/////////////////////////////////////////////////////////////////////////////////////MACHINE STATUS/////////////////////////////////////////////////////////////////////////////////////
stMachineStatus.bSystemPowerUp 			:= (stMachineStatus.eMachineState = E_MachineState.SYSTEM_POWER_UP);
stMachineStatus.bStopped 				:= (stMachineStatus.eMachineState = E_MachineState.STOPPED);
stMachineStatus.bInitialising 			:= (stMachineStatus.eMachineState = E_MachineState.SYSTEM_INITIALISING);
stMachineStatus.bReadyToStart 			:= (stMachineStatus.eMachineState = E_MachineState.SYSTEM_READY_TO_START);
stMachineStatus.bAutoCycle 				:= (stMachineStatus.eMachineState = E_MachineState.SYSTEM_AUTO_CYCLE);
stMachineStatus.bStopping 				:= (stMachineStatus.eMachineState = E_MachineState.STOPPING);
stMachineStatus.bFault 					:= (stMachineStatus.eMachineState = E_MachineState.FAULT);
stMachineStatus.bManualMode 			:= (stMachineStatus.eMachineState = E_MachineState.MANUAL_MODE);
stMachineStatus.bSafety 				:= (stMachineStatus.eMachineState = E_MachineState.SAFETY);

/////////////////////////////////////////////////////////////////////////////////////FLAGS/////////////////////////////////////////////////////////////////////////////////////
stMasterCtrl.bAllStationsStopped		:= (stCamera.Status.bStopped OR NOT stMACHINE.bVisionTest ) AND (stLeakTesters.Status.bStopped OR NOT stMACHINE.bLeakTest ) AND (stHeightTests.Status.bStopped OR NOT stMACHINE.bHeightTest ) AND stProcessCylinder.Status.bStopped AND stProcessDoor.Status.bStopped AND
										   (NOT stCamera.Status.bBusy OR NOT stMACHINE.bVisionTest ) AND (NOT stLeakTesters.Status.bBusy OR NOT stMACHINE.bLeakTest ) AND (NOT stHeightTests.Status.bBusy OR NOT stMACHINE.bHeightTest ) AND NOT stProcessCylinder.Status.bBusy AND NOT stProcessDoor.Status.bBusy;
										   
stMasterCtrl.bAllStationsReady			:= (stCamera.Status.bReady OR NOT stMACHINE.bVisionTest ) AND (stLeakTesters.Status.bReady OR NOT stMACHINE.bLeakTest ) AND (stHeightTests.Status.bReady OR NOT stMACHINE.bHeightTest ) AND stProcessCylinder.Status.bReady AND stProcessDoor.Status.bReady;
END_ACTION

ACTION b_ACT_ProcessCycle:
/////////////////////////////////////////////////////////////////////////////////////UTILITIES & TRIGGERS/////////////////////////////////////////////////////////////////////////////////////
//ADD REJECT SENSOR FUNCTION. IF PART FAIL WE SHOULD WAIT UNTIL THE OPERATOR LEAVE THE FAIL PART IN THE CONTAINER
tonTakePicture(IN := stCamera.Status.bDone, PT := T#500MS);

ctuRejectPart();
IF eCycleState = E_General_ProcessCycle.RESET_ALL_CMD THEN
	
	ctuRejectPart.RESET							:= TRUE;

ELSE ctuRejectPart.RESET						:= FALSE;	
	
END_IF
IF eCycleState = E_General_ProcessCycle.IDLE THEN
	
	bAutocycleIDLE								:= TRUE;
	
ELSE bAutocycleIDLE								:= FALSE;

END_IF

tonWaitExtendCylidner(IN := eCycleState = E_General_ProcessCycle.PROCESS_FLAGS_DEFINITIONS, PT := T#1S);
tonGettingResults( IN := eCycleState = E_General_ProcessCycle.WAIT_RESULTS, PT := T#100MS);

tonCMD_Done( IN := , PT := T#500MS);
tonSave_Data( IN :=  eCycleState = E_General_ProcessCycle.SAVE_DATA2, PT := T#500MS);
tonResetAllCMD( IN := eCycleState = E_General_ProcessCycle.RESET_ALL_CMD, PT := T#500MS);


tonExecute( IN := 	eCycleState = E_General_ProcessCycle.CLOSE_PROCESS_DOOR OR
					eCycleState = E_General_ProcessCycle.OPEN_PROCESS_DOOR OR
					eCycleState = E_General_ProcessCycle.WAIT_PRE_RETRACT_PROCESS_CYLINDER OR
					eCycleState = E_General_ProcessCycle.EXTEND_PROCESS_CYLINDER OR
					eCycleState = E_General_ProcessCycle.RETRACT_PROCESS_CYLINDER OR
					eCycleState = E_General_ProcessCycle.CAMERA_INSPECTION OR
					eCycleState = E_General_ProcessCycle.LEAK_TESTS OR
					eCycleState = E_General_ProcessCycle.LEAK_TESTS_HEIGHT_TEST OR
					eCycleState = E_General_ProcessCycle.HEIGHT_TEST OR
					eCycleState = E_General_ProcessCycle.WAIT_TO_SAVE_DATA,
					PT := T#500MS);
					
tonCylinderDwell( IN := eCycleState = E_General_ProcessCycle.PRE_RETRACT_PROCESS_CYLINDER, PT := T#250MS);

IF (stMachineStatus.eMachineState <> E_MachineState.SYSTEM_AUTO_CYCLE) THEN
	
	eCycleState												:= E_General_ProcessCycle.RESET_ALL_CMD;

END_IF

rFirstAutoCycle( CLK := stMachineStatus.bAutoCycle);

IF (eCycleState = E_General_ProcessCycle.CAMERA_INSPECTION) OR (eCycleState = E_General_ProcessCycle.LEAK_TESTS) OR
	(eCycleState = E_General_ProcessCycle.LEAK_TESTS_HEIGHT_TEST) OR (eCycleState = E_General_ProcessCycle.HEIGHT_TEST)  THEN
			sMachineMessage						:= 'Inspection in process';

END_IF

IF stMachineStatus.eMachineState <> E_MachineState.SYSTEM_AUTO_CYCLE THEN
	
	MEMSET( destAddr := ADR(stCycleDataNest1), fillByte := 0, n := SIZEOF(stCycleDataNest1));
	MEMSET( destAddr := ADR(stCycleDataNest2), fillByte := 0, n := SIZEOF(stCycleDataNest2));

END_IF

(* Renan Added 10Jul26*)
bPuckLockerEnable := GVL_Master.stMACHINE.bMachine[2] AND GVL_HMI.bPuckLockerGateEnable;
(*\Renan Added 10Jul26*)

(*Renan added - Puck Locker Bug - 08Jul26*)
bPuckLockerReadyToStart := (NOT bPuckLockerEnable) OR (GVL_Stations.stPuckLocker.bPuckDetected AND
							GVL_Stations.stPuckLocker.bPuckLocked AND GVL_Stations.stPuckLocker.eState = E_PuckLockerState.Locked);
(*\Renan added - Puck Locker Bug - 08Jul26*)

(*Renan Added 06Jul26*)
IF bPuckLockerEnable THEN
	GVL_Stations.stPuckLocker.bNestsEmpty := ((NOT bProcessedPart[0]) OR (NOT bPartPresentNest1)) AND ((NOT bProcessedPart[1]) OR (NOT bPartPresentNest2));
ELSE
	GVL_Stations.stPuckLocker.bNestsEmpty := TRUE;
END_IF
(*\Renan Added 06Jul26*)



/////////////////////////////////////////////////////////////////////////////////////CONDITIONS/////////////////////////////////////////////////////////////////////////////////////

(* Renan Added - Buglist n6 - 08Jul26 *)
bNest1StartOK := (NOT bNest1Flag) OR bPartPresentNest1;
bNest2StartOK := (NOT bNest2Flag) OR bPartPresentNest2;
(*\Renan Added - Buglist n6 - 08Jul26 *)

bStartProcessCondition := bTwoHandsSignal AND bPartPresentNest1 AND bPartPresentNest2 AND (bNest1Flag OR bNest2Flag);

IF rFirstAutoCycle.Q THEN
	eCycleState												:= E_General_ProcessCycle.RESET_ALL_CMD;
END_IF


CASE eCycleState OF
	
E_General_ProcessCycle.RESET_ALL_CMD:

				stProcessDoor.CMD.ProcessDoorCMD.OpenDoor						:= FALSE;
				stProcessDoor.CMD.ProcessDoorCMD.CloseDoor						:= FALSE;
				stProcessDoor.CMD.bExecute										:= FALSE;
				
				stProcessCylinder.CMD.ProcessCylinderCMD.ExtendCylinder1		:= FALSE;
				stProcessCylinder.CMD.ProcessCylinderCMD.RetractCylinder1		:= FALSE;
				stProcessCylinder.CMD.bExecute									:= FALSE;
				
				stLeakTesters.CMD.LeakTestersCMD.RunLeakTester1					:= FALSE;
				stLeakTesters.CMD.LeakTestersCMD.RunLeakTester2					:= FALSE;
				stLeakTesters.CMD.bExecute										:= FALSE;
				
				stHeightTests.CMD.HeightTest_CMD.Measurement1					:= FALSE;
				stHeightTests.CMD.HeightTest_CMD.Measurement2					:= FALSE;
				stHeightTests.CMD.bExecute										:= FALSE;
				
				stCamera.CMD.bExecute											:= FALSE;
				
				bVisionProcessDoneFlag											:= FALSE;
				
				bWriteNest1														:= FALSE;
				bWriteNest2														:= FALSE;
				bRejectPartDialog[0]											:= FALSE;
				bRejectPartDialog[1]											:= FALSE;
				bRejectPartFault												:= FALSE;
				
				bProcessedPart[0]												:= FALSE;
				bProcessedPart[1]												:= FALSE;
			
				//add reset command to reset all cycle data
				
				IF tonResetAllCMD.Q AND stMachineStatus.bAutoCycle THEN
					eCycleState								:= E_General_ProcessCycle.IDLE;						
				END_IF
	
E_General_ProcessCycle.IDLE:

				//start cycle
				IF bStartProcessCondition AND bPartPresent[0] AND bPartPresent[1] AND bPuckLockerReadyToStart THEN (*Renan added - Puck Locker Bug - 08Jul26*) //Original: IF bStartProcessCondition AND NOT bProcessedPart[0] AND NOT bProcessedPart[1] THEN
					
					MEMSET( destAddr := ADR(stCycleDataNest1), fillByte := 0, n := SIZEOF(stCycleDataNest1));
					MEMSET( destAddr := ADR(stCycleDataNest2), fillByte := 0, n := SIZEOF(stCycleDataNest2));
					
					IF bNest1Flag THEN
						
						bProcessedPart[0]					:= bPartPresentNest1;
						
					END_IF
					
					IF bNest2Flag THEN
						
						bProcessedPart[1]					:= bPartPresentNest2;
						
					END_IF
					
					eCycleState								:= E_General_ProcessCycle.CLOSE_PROCESS_DOOR;
					
				END_IF
				
				IF bPuckLockerEnable AND NOT bPuckLockerReadyToStart AND NOT bProcessedPart[0] AND NOT bProcessedPart[1] THEN
				
					IF NOT GVL_Stations.stPuckLocker.bPuckDetected THEN
						
						sMachineMessage 		:= 'Insert puck into locker to continue';
						
					ELSE
						
						sMachineMessage := 'Waiting for puck locker to lock puck';
						
					END_IF					
				
				ELSIF  bPuckLockerReadyToStart AND bPartPresent[0] AND bPartPresent[1] THEN
					
					sMachineMessage := 'trigger both safety buttons to start cycle';
					
				ELSIF bPuckLockerReadyToStart AND ( NOT bPartPresent[0] AND NOT bPartPresent[1]) THEN
					
					sMachineMessage 			:= 'Place parts to continue';
					
				ELSIF bPuckLockerReadyToStart AND ( bPartPresent[0] AND NOT bPartPresent[1]) THEN
					
					sMachineMessage 			:= 'Place part in nest 2 to continue';
				
				ELSIF bPuckLockerReadyToStart AND ( NOT bPartPresent[0] AND bPartPresent[1]) THEN
					
					sMachineMessage 			:= 'Place part in nest 1 to continue';
					
				END_IF
			
E_General_ProcessCycle.CLOSE_PROCESS_DOOR:

				stProcessDoor.CMD.ProcessDoorCMD.CloseDoor	:= TRUE;
				stProcessDoor.CMD.bExecute					:= TRUE;
				
				IF tonExecute.Q THEN
					eCycleState								:= E_General_ProcessCycle.WAIT_CLOSE_PROCESS_DOOR;	
				END_IF

E_General_ProcessCycle.WAIT_CLOSE_PROCESS_DOOR:
				
				IF stProcessDoor.Status.bDone THEN
				stProcessDoor.CMD.ProcessDoorCMD.CloseDoor	:= FALSE;
				stProcessDoor.CMD.bExecute					:= FALSE;
				stProcessDoor.CMD.bAcknowledge				:= TRUE;
				eCycleState									:= E_General_ProcessCycle.PROCESS_FLAGS_DEFINITIONS;
				END_IF
				
E_General_ProcessCycle.PROCESS_FLAGS_DEFINITIONS:
				
				
				IF stMACHINE.bVisionTest THEN
					
					IF bVisionProcessDoneFlag THEN
						
						eCycleState							:= E_General_ProcessCycle.PRE_RETRACT_PROCESS_CYLINDER; //Renan changed - Buglist n13 08Jul26 | Original: \\E_General_ProcessCycle.EXTEND_PROCESS_CYLINDER;
					ELSE eCycleState						:= E_General_ProcessCycle.CAMERA_INSPECTION;
						
					END_IF
				ELSIF tonWaitExtendCylidner.Q AND NOT stMACHINE.bVisionTest THEN

					eCycleState							:= E_General_ProcessCycle.PRE_RETRACT_PROCESS_CYLINDER; //Renan changed - Buglist n13 08Jul26 | Original: \\E_General_ProcessCycle.EXTEND_PROCESS_CYLINDER;
					
				END_IF
				
(* Renan added - Buglist n13 - 08Jul26 *)				
E_General_ProcessCycle.PRE_RETRACT_PROCESS_CYLINDER:		

				stProcessCylinder.CMD.ProcessCylinderCMD.RetractCylinder1		:= TRUE;	
				stProcessCylinder.CMD.bExecute			:= TRUE;
				
				IF tonCylinderDwell.Q THEN
					eCycleState							:= E_General_ProcessCycle.WAIT_PRE_RETRACT_PROCESS_CYLINDER;	
				END_IF

E_General_ProcessCycle.WAIT_PRE_RETRACT_PROCESS_CYLINDER:

				IF 	stProcessCylinder.Status.bDone OR stProcessCylinder.Status.bReady THEN
					
					stProcessCylinder.CMD.ProcessCylinderCMD.RetractCylinder1		:= FALSE;
					stProcessCylinder.CMD.bExecute		:= FALSE;
					stProcessCylinder.CMD.bAcknowledge	:= TRUE;
					
					IF tonExecute.Q THEN
						eCycleState							:= E_General_ProcessCycle.EXTEND_PROCESS_CYLINDER;
					END_IF	
				END_IF
(*\Renan added - Buglist n13 - 08Jul26 *)

E_General_ProcessCycle.EXTEND_PROCESS_CYLINDER:
				
						
				stProcessCylinder.CMD.ProcessCylinderCMD.ExtendCylinder1		:= TRUE;
				stProcessCylinder.CMD.bExecute		:= TRUE;
	
				IF tonExecute.Q THEN
					eCycleState								:= E_General_ProcessCycle.WAIT_EXTEND_PROCESS_CYLINDER;	
				END_IF

E_General_ProcessCycle.WAIT_EXTEND_PROCESS_CYLINDER:
			
				IF stProcessCylinder.Status.bDone THEN
					
					stProcessCylinder.CMD.ProcessCylinderCMD.ExtendCylinder1		:= FALSE;
					stProcessCylinder.CMD.bExecute			:= FALSE;
					stProcessCylinder.CMD.bAcknowledge		:= TRUE;
						
					IF stMACHINE.bHeightTest AND stMACHINE.bLeakTest THEN
						
						eCycleState							:= E_General_ProcessCycle.LEAK_TESTS_HEIGHT_TEST;	
						
					ELSIF 	stMACHINE.bHeightTest AND NOT stMACHINE.bLeakTest  THEN
						
						eCycleState							:= E_General_ProcessCycle.HEIGHT_TEST;
					
					ELSIF 	NOT stMACHINE.bHeightTest AND stMACHINE.bLeakTest  THEN
						
						eCycleState							:= E_General_ProcessCycle.LEAK_TESTS;
					END_IF
					
				END_IF

E_General_ProcessCycle.LEAK_TESTS_HEIGHT_TEST:
				
							
				stLeakTesters.CMD.LeakTestersCMD.RunLeakTester1						:= bNest1Flag;
				stLeakTesters.CMD.LeakTestersCMD.RunLeakTester2						:= bNest2Flag;
				stHeightTests.CMD.HeightTest_CMD.Measurement1						:= bNest1Flag;
				stHeightTests.CMD.HeightTest_CMD.Measurement2						:= bNest2Flag;
				stLeakTesters.CMD.bExecute					:= TRUE;
				stHeightTests.CMD.bExecute					:= TRUE;
							
				IF tonExecute.Q THEN
					eCycleState								:= E_General_ProcessCycle.WAIT_LEAK_TEST_HEIGHT_TEST;	
				END_IF

E_General_ProcessCycle.WAIT_LEAK_TEST_HEIGHT_TEST:
					
					IF stLeakTesters.Status.bDone AND stHeightTests.Status.bDone THEN
						
						stLeakTesters.CMD.LeakTestersCMD.RunLeakTester1				:= FALSE;
						stLeakTesters.CMD.LeakTestersCMD.RunLeakTester2				:= FALSE;
						stHeightTests.CMD.HeightTest_CMD.Measurement1				:= FALSE;
						stHeightTests.CMD.HeightTest_CMD.Measurement2				:= FALSE;
						stLeakTesters.CMD.bExecute			:= FALSE;
						stHeightTests.CMD.bExecute			:= FALSE;
						stLeakTesters.CMD.bAcknowledge		:= TRUE;
						stHeightTests.CMD.bAcknowledge		:= TRUE;
						eCycleState							:= E_General_ProcessCycle.WAIT_RESULTS;
						
					END_IF				   

E_General_ProcessCycle.HEIGHT_TEST:

				stHeightTests.CMD.HeightTest_CMD.Measurement1				 		:= bNest1Flag;
				stHeightTests.CMD.HeightTest_CMD.Measurement2				 		:= bNest2Flag;
				stHeightTests.CMD.bExecute					:= TRUE;
					
				IF tonExecute.Q THEN
					eCycleState								:= E_General_ProcessCycle.WAIT_HEIGHT_TEST;	
				END_IF

E_General_ProcessCycle.WAIT_HEIGHT_TEST:

				IF stHeightTests.Status.bDone THEN
					
					stHeightTests.CMD.HeightTest_CMD.Measurement1				 	:= FALSE;
					stHeightTests.CMD.HeightTest_CMD.Measurement2				 	:= FALSE;
					stHeightTests.CMD.bExecute										:= FALSE;
					stHeightTests.CMD.bAcknowledge 			:= TRUE;	
					eCycleState								:= E_General_ProcessCycle.WAIT_RESULTS;
					
				END_IF

E_General_ProcessCycle.LEAK_TESTS:

				stLeakTesters.CMD.LeakTestersCMD.RunLeakTester1						:= bNest1Flag;
				stLeakTesters.CMD.LeakTestersCMD.RunLeakTester2						:= bNest2Flag;
				stLeakTesters.CMD.bExecute					:= TRUE;
				
				IF tonExecute.Q THEN
					eCycleState								:= E_General_ProcessCycle.WAIT_LEAK_TEST;	
				END_IF

E_General_ProcessCycle.WAIT_LEAK_TEST:

				IF stLeakTesters.Status.bDone THEN
					
					stLeakTesters.CMD.bExecute										:= FALSE;
					stLeakTesters.CMD.LeakTestersCMD.RunLeakTester1				 	:= FALSE;
					stLeakTesters.CMD.LeakTestersCMD.RunLeakTester2				 	:= FALSE;
					stLeakTesters.CMD.bAcknowledge 			:= TRUE;	
					eCycleState								:= E_General_ProcessCycle.WAIT_RESULTS;
					
				END_IF
				
E_General_ProcessCycle.CAMERA_INSPECTION:
				
				stCamera.CMD.bExecute						:= TRUE;
				stCamera.CMD.CameraCMD.Inspect1				:= bNest1Flag;
				stCamera.CMD.CameraCMD.Inspect2				:= bNest2Flag;
				
				IF tonExecute.Q THEN
					eCycleState								:= E_General_ProcessCycle.WAIT_CAMERA;	
				END_IF
				
E_General_ProcessCycle.WAIT_CAMERA:

				IF  tonTakePicture.Q THEN
					
					stCamera.CMD.bExecute					:= FALSE;
					bVisionProcessDoneFlag					:= TRUE;
					stCamera.CMD.bAcknowledge				:= TRUE;
					eCycleState								:= E_General_ProcessCycle.PROCESS_FLAGS_DEFINITIONS;
				
				END_IF
				
E_General_ProcessCycle.WAIT_RESULTS:

				IF tonGettingResults.Q THEN
					
					eCycleState									:= E_General_ProcessCycle.RESULTS;
					
				END_IF


E_General_ProcessCycle.RESULTS:

				
					
					IF bProcessedPart[0] THEN
					
						IF  (stCycleDataNest1.Camera_Pass OR NOT stMACHINE.bVisionTest) AND   (stCycleDataNest1.LeakTest_Pass OR NOT stMACHINE.bLeakTest)
				 			AND   (stCycleDataNest1.HeightTest_Pass OR NOT stMACHINE.bHeightTest) THEN	
				
							stCycleDataNest1.bPass				:= TRUE;
							stCycleDataNest1.bFail				:= FALSE;
				
						ELSE stCycleDataNest1.bFail				:= TRUE;
							stCycleDataNest1.bPass				:= FALSE;
				
						END_IF
					
					END_IF
				
					IF bProcessedPart[1] THEN
					
						IF  (stCycleDataNest2.Camera_Pass OR NOT stMACHINE.bVisionTest) AND   (stCycleDataNest2.LeakTest_Pass OR NOT stMACHINE.bLeakTest)
				 			AND   (stCycleDataNest2.HeightTest_Pass OR NOT stMACHINE.bHeightTest) THEN	
				
							stCycleDataNest2.bPass				:= TRUE;
							stCycleDataNest2.bFail				:= FALSE;
				
						ELSE stCycleDataNest2.bFail				:= TRUE;
							stCycleDataNest2.bPass				:= FALSE;
				
						END_IF
					
					END_IF
					
				
				
				
				
				stCycleDataNest1.sTime						:= sSystemTime;
				stCycleDataNest1.sDate						:= sSystemDate;
				stCycleDataNest2.sTime						:= sSystemTime;
				stCycleDataNest2.sDate						:= sSystemDate;
					
				eCycleState								:= E_General_ProcessCycle.WAIT_TO_SAVE_DATA;
									
E_General_ProcessCycle.WAIT_TO_SAVE_DATA:
				
				IF tonExecute.Q THEN
					eCycleState								:= E_General_ProcessCycle.SAVE_DATA;	
				END_IF

E_General_ProcessCycle.SAVE_DATA:

				IF bProcessedPart[0] THEN
					
					FOR i := 199 TO 0 BY -1 DO
						aDataHistoryNest1[i+1] 						:= aDataHistoryNest1[i];
					END_FOR
				
				END_IF
				
				IF bProcessedPart[1] THEN
					
					FOR i := 199 TO 0 BY -1 DO
						aDataHistoryNest2[i+1] 						:= aDataHistoryNest2[i];
					END_FOR
				
				END_IF		
			
				eCycleState									:= E_General_ProcessCycle.SAVE_DATA2;
					
E_General_ProcessCycle.SAVE_DATA2:	
				
				
				c_ACT_SaveData();	
				
				
					
				eCycleState									:= E_General_ProcessCycle.CSV_NEST1;
				
				
E_General_ProcessCycle.CSV_NEST1:

				IF bProcessedPart[0] THEN
					
					bWriteNest1								:= TRUE;
					
					IF bCSVDone OR bCSVError THEN
						
						eCycleState							:= E_General_ProcessCycle.CSV_NEST2;
						bWriteNest1							:= FALSE;
						bCSVError							:= FALSE;
						
					END_IF
				ELSE eCycleState							:= E_General_ProcessCycle.CSV_NEST2;				
					
				END_IF
			
				
E_General_ProcessCycle.CSV_NEST2:

				IF bCSVDone THEN
					
						bWriteNest2							:= FALSE;
						eCycleState							:= E_General_ProcessCycle.RETRACT_PROCESS_CYLINDER;	
	
				END_IF

				IF bProcessedPart[1] AND  bCSVReady AND NOT bCSVDone AND NOT bCSVError THEN
				
						bWriteNest2							:= TRUE;

				ELSIF NOT bProcessedPart[1] OR bCSVError THEN

						 eCycleState						:= E_General_ProcessCycle.RETRACT_PROCESS_CYLINDER;
						 bCSVError							:= FALSE;
						 
				END_IF
				
				
					
				
E_General_ProcessCycle.RETRACT_PROCESS_CYLINDER:
						
				stProcessCylinder.CMD.ProcessCylinderCMD.RetractCylinder1		:= TRUE;	
				stProcessCylinder.CMD.bExecute			:= TRUE;
				
				IF tonExecute.Q THEN
					eCycleState							:= E_General_ProcessCycle.WAIT_RETRACT_PROCESS_CYLINDER;	
				END_IF

E_General_ProcessCycle.WAIT_RETRACT_PROCESS_CYLINDER:

				IF 	stProcessCylinder.Status.bDone THEN
					
					stProcessCylinder.CMD.ProcessCylinderCMD.RetractCylinder1		:= FALSE;
					stProcessCylinder.CMD.bExecute		:= FALSE;
					stProcessCylinder.CMD.bAcknowledge	:= TRUE;
					
					IF NOT bEmptyRejectChute THEN

						eCycleState							:= E_General_ProcessCycle.OPEN_PROCESS_DOOR;
					
					ELSE eCycleState							:= E_General_ProcessCycle.REJECT_CHUTE_FULL; 
					
					END_IF
					
				END_IF
		
E_General_ProcessCycle.REJECT_CHUTE_FULL:

				sMachineMessage									:= 'Waiting for Reject chute empty';

				IF NOT bEmptyRejectChute THEN
					
						sMachineMessage							:= '';
						eCycleState								:= E_General_ProcessCycle.OPEN_PROCESS_DOOR;
				
				END_IF	
		
E_General_ProcessCycle.OPEN_PROCESS_DOOR:

				stProcessDoor.CMD.ProcessDoorCMD.OpenDoor							:= TRUE;
				stProcessDoor.CMD.bExecute				:= TRUE;
				
				IF tonExecute.Q THEN
					eCycleState							:= E_General_ProcessCycle.WAIT_OPEN_PROCESS_DOOR;	
				END_IF

E_General_ProcessCycle.WAIT_OPEN_PROCESS_DOOR:

				IF 	stProcessDoor.Status.bDone THEN
					
					stProcessDoor.CMD.ProcessDoorCMD.OpenDoor						:= FALSE;
					stProcessDoor.CMD.bExecute			:= FALSE;
					stProcessDoor.CMD.bAcknowledge		:= TRUE;
					
					eCycleState							:= E_General_ProcessCycle.PUCK_DEFINITION;
					
				END_IF
				
E_General_ProcessCycle.PUCK_DEFINITION:
		
				(* Renan Added - Buglist n6 - 08Jul26 *)
				bCycleHasFailure := (bProcessedPart[0] AND stCycleDataNest1.bFail) OR (bProcessedPart[1] AND stCycleDataNest2.bFail);

				bCycleAllProcessedPass := (bProcessedPart[0] OR bProcessedPart[1]) AND ((NOT bProcessedPart[0]) OR stCycleDataNest1.bPass) AND ((NOT bProcessedPart[1]) OR stCycleDataNest2.bPass);
					(*\Renan Added - Buglist n6 - 08Jul26 *)
					
					(* Renan Added 10Jul26 - Puck Locker *)
				IF bPuckLockerEnable AND bCycleAllProcessedPass THEN
					
					GVL_Stations.stPuckLocker.nRequestedRelease := USINT#0;
					
					IF bProcessedPart[0] AND stCycleDataNest1.bPass THEN
						
						GVL_Stations.stPuckLocker.nRequestedRelease := GVL_Stations.stPuckLocker.nRequestedRelease + USINT#1;
						
					END_IF
					
					IF bProcessedPart[1] AND stCycleDataNest2.bPass THEN
						
						GVL_Stations.stPuckLocker.nRequestedRelease := GVL_Stations.stPuckLocker.nRequestedRelease + USINT#1;
							
					END_IF
					
					GVL_Stations.stPuckLocker.bApplyDisposition := TRUE;
					
				END_IF
				
				
				IF bCycleHasFailure THEN //Bugfix 08Jul26
					
					eCycleState								:= E_General_ProcessCycle.WAIT_REJECT_PART;
					
				ELSIF bCycleAllProcessedPass THEN //Bugfix 08Jul26

					eCycleState								:= E_General_ProcessCycle.NEST_CLEARING;
						
				END_IF		
			
E_General_ProcessCycle.WAIT_REJECT_PART:
					
				ctuRejectPart.CU 								:= rRejectSensor.Q;				

				IF stCycleDataNest1.bFail AND NOT stCycleDataNest2.bFail THEN
					
					sMachineMessage												:= 'REMOVE PART FROM NEST 1 AND PUT IN REJECT CHUTE';
					
					IF ctuRejectPart.CV > 0 AND NOT bPartPresentNest1 AND (bPartPresentNest2 OR NOT bProcessedPart[1])  THEN
						
						(* Renan Added 10Jul26 - Puck Locker *)
						IF bPuckLockerEnable THEN
							GVL_Stations.stPuckLocker.nRequestedRelease 		:= USINT#1;
							GVL_Stations.stPuckLocker.bApplyDisposition 		:= TRUE;
						END_IF
						(*\Renan Added 10Jul26 - Puck Locker *)
						
						eCycleState												:= E_General_ProcessCycle.NEST_CLEARING;
						
					ELSIF ctuRejectPart.CV > 0 AND (bPartPresentNest1 OR (NOT bPartPresentNest2 AND bProcessedPart[1])) THEN
						
						bRejectPartFault										:= TRUE; 
					
					END_IF
					
					IF NOT bPartPresentNest2 AND bProcessedPart[1] THEN
						
						bRejectPartDialog[0]									:= TRUE;		
						sMachineMessage											:= 'WRONG PART TAKEN';
						
					ELSIF  bPartPresentNest2 THEN
						
						bRejectPartDialog[0]									:= FALSE;
						
					END_IF					
					
				ELSIF NOT stCycleDataNest1.bFail AND stCycleDataNest2.bFail THEN
					
					sMachineMessage												:= 'REMOVE PART FROM NEST 2 AND PUT IN REJECT CHUTE';
					
					IF ctuRejectPart.CV > 0 AND NOT bPartPresentNest2 AND (bPartPresentNest1 OR NOT bProcessedPart[0])  THEN
						
						(* Renan Added 10Jul26 - Puck Locker *)
						IF bPuckLockerEnable THEN
							GVL_Stations.stPuckLocker.nRequestedRelease 		:= USINT#1;
							GVL_Stations.stPuckLocker.bApplyDisposition 		:= TRUE;
						END_IF
						(*\Renan Added 10Jul26 - Puck Locker *)
						
						
						eCycleState												:= E_General_ProcessCycle.NEST_CLEARING;
						
					ELSIF ctuRejectPart.CV > 0 AND (bPartPresentNest1 OR (NOT bPartPresentNest1 AND bProcessedPart[0])) THEN
						
						bRejectPartFault										:= TRUE; 
					
					END_IF
					
					IF NOT bPartPresentNest1 AND bProcessedPart[0] THEN
						
						bRejectPartDialog[1]									:= TRUE;		
						sMachineMessage											:= 'WRONG PART TAKEN';
						
					ELSIF  bPartPresentNest1 THEN
						
						bRejectPartDialog[1]									:= FALSE;
						
					END_IF
				
				ELSIF stCycleDataNest1.bFail AND stCycleDataNest2.bFail THEN
					
					IF ctuRejectPart.CV > 1 AND NOT bPartPresentNest1 AND NOT bPartPresentNest2 THEN
						
						(* Renan Added 10Jul26 - Puck Locker *)
						IF bPuckLockerEnable THEN
							GVL_Stations.stPuckLocker.nRequestedRelease 		:= USINT#0;
							GVL_Stations.stPuckLocker.bApplyDisposition 		:= TRUE;
						END_IF
						(*\Renan Added 10Jul26 - Puck Locker *)
						
						eCycleState												:= E_General_ProcessCycle.NEST_CLEARING;
					
					ELSIF ctuRejectPart.CV > 1 AND ( bPartPresentNest1 OR bPartPresentNest2) THEN
						
						bRejectPartFault										:= TRUE; 		
					
					END_IF;
					
					sMachineMessage												:= 'REMOVE PART FROM BOTH NESTS AND PUT IN REJECT CHUTE';
					
				END_IF
				
E_General_ProcessCycle.NEST_CLEARING:
				
				IF bPuckLockerEnable AND GVL_Stations.stPuckLocker.eState = E_PuckLockerState.WaitingForNestsEmpty THEN
				
					IF (bPartPresentNest1 AND bNest1Flag) OR (bPartPresentNest2 AND bNest2Flag) THEN
						
						sMachineMessage 										:= 'Remove parts from nests to release puck';
						
					ELSE
						
						sMachineMessage 										:= 'Waiting for puck to be released';
						
					END_IF
				
				ELSIF (bPartPresentNest1 AND bNest1Flag) AND NOT (bPartPresentNest2 AND bNest2Flag)  THEN
					
					IF bPuckLockerEnable THEN
						
						sMachineMessage 										:= 'Remove processed part from nest 1 to release puck';
						
					ELSE
						
						sMachineMessage 										:= 'Remove Processed part from nest 1';
						
					END_IF
					
				ELSIF NOT (bPartPresentNest1 AND bNest1Flag) AND (bPartPresentNest2 AND bNest2Flag)  THEN 
					
					IF bPuckLockerEnable THEN
						
						sMachineMessage 										:= 'Remove processed part from nest 2 to release puck';
						
					ELSE
						
						sMachineMessage 										:= 'Remove Processed part from nest 2';
						
					END_IF
					
				ELSIF (bPartPresentNest1 AND bNest1Flag) AND (bPartPresentNest2 AND bNest2Flag) THEN 
					
					IF bPuckLockerEnable THEN
						
						sMachineMessage 										:= 'Remove processed parts to release puck';
						
					ELSE
						
						sMachineMessage 										:= 'Remove Processed parts';
						
					END_IF
					
				ELSIF (NOT bPartPresentNest1 OR NOT bNest1Flag) AND (NOT bPartPresentNest2 OR NOT bNest2Flag)  THEN
					
					sMachineMessage 											:= '';
					eCycleState													:= E_General_ProcessCycle.RESET_ALL_CMD;
									
				END_IF
				
END_CASE
END_ACTION

ACTION c_ACT_SaveData:

//SAVING NEST 1 DATA
IF bProcessedPart[0] THEN
	
	stCycleDataNest1.sDistance1				:= REAL_TO_STRING(stCycleDataNest1.HeightTest_anDistancesResult[1]);
	stCycleDataNest1.sDistance2				:= REAL_TO_STRING(stCycleDataNest1.HeightTest_anDistancesResult[2]);
	stCycleDataNest1.sDistance3				:= REAL_TO_STRING(stCycleDataNest1.HeightTest_anDistancesResult[3]);
	
	stCycleDataNest1.sSetpoint1				:= REAL_TO_STRING(stCycleDataNest1.HeightTest_anSetPoint[1]);
	stCycleDataNest1.sSetpoint2				:= REAL_TO_STRING(stCycleDataNest1.HeightTest_anSetPoint[2]);
	stCycleDataNest1.sSetpoint3				:= REAL_TO_STRING(stCycleDataNest1.HeightTest_anSetPoint[3]);
	
	IF stCycleDataNest1.bPass THEN
	
		stCycleDataNest1.sGeneralResult			:= 'PASS';

	ELSIF stCycleDataNest1.bFail THEN
	
		stCycleDataNest1.sGeneralResult			:= 'FAIL';

	END_IF
	


	IF stCycleDataNest1.Camera_Pass THEN
	
		stCycleDataNest1.sCameraResult			:= 'PASS';

	ELSIF stCycleDataNest1.Camera_Fail THEN
	
		stCycleDataNest1.sCameraResult			:= 'FAIL';

	END_IF

	IF stCycleDataNest1.HeightTest_Pass THEN
	
		stCycleDataNest1.sHeightTestResult		:= 'PASS';
	
	ELSIF stCycleDataNest1.HeightTest_Fail THEN
	
		stCycleDataNest1.sHeightTestResult		:= 'FAIL';
	
	END_IF



	IF stCycleDataNest1.LeakTest_Pass THEN
	
		stCycleDataNest1.sLeakTesterResult		:= 'PASS';

	ELSIF stCycleDataNest1.LeakTest_Fail THEN
	
		stCycleDataNest1.sLeakTesterResult		:= 'FAIL';
	
	END_IF
	
	aDataHistoryNest1[0]						:= stCycleDataNest1;
	
END_IF;
	

//SAVING NEST 2 DATA

IF bProcessedPart[1] THEN
	
	stCycleDataNest2.sDistance1				:= REAL_TO_STRING(stCycleDataNest2.HeightTest_anDistancesResult[1]);
	stCycleDataNest2.sDistance2				:= REAL_TO_STRING(stCycleDataNest2.HeightTest_anDistancesResult[2]);
	stCycleDataNest2.sDistance3				:= REAL_TO_STRING(stCycleDataNest2.HeightTest_anDistancesResult[3]);
	
	stCycleDataNest2.sSetpoint1				:= REAL_TO_STRING(stCycleDataNest2.HeightTest_anSetPoint[1]);
	stCycleDataNest2.sSetpoint2				:= REAL_TO_STRING(stCycleDataNest2.HeightTest_anSetPoint[2]);
	stCycleDataNest2.sSetpoint3				:= REAL_TO_STRING(stCycleDataNest2.HeightTest_anSetPoint[3]);
	
	IF stCycleDataNest2.bPass THEN
	
		stCycleDataNest2.sGeneralResult			:= 'PASS';

	ELSIF stCycleDataNest2.bFail THEN
	
		stCycleDataNest2.sGeneralResult			:= 'FAIL';

	END_IF
	


	IF stCycleDataNest2.Camera_Pass THEN
	
		stCycleDataNest2.sCameraResult			:= 'PASS';

	ELSIF stCycleDataNest2.Camera_Fail THEN
	
		stCycleDataNest2.sCameraResult			:= 'FAIL';

	END_IF

	IF stCycleDataNest2.HeightTest_Pass THEN
	
		stCycleDataNest2.sHeightTestResult		:= 'PASS';
	
	ELSIF stCycleDataNest2.HeightTest_Fail THEN
	
		stCycleDataNest2.sHeightTestResult		:= 'FAIL';
	
	END_IF



	IF stCycleDataNest2.LeakTest_Pass THEN
	
		stCycleDataNest2.sLeakTesterResult		:= 'PASS';

	ELSIF stCycleDataNest2.LeakTest_Fail THEN
	
		stCycleDataNest2.sLeakTesterResult		:= 'FAIL';
	
	END_IF
	
	aDataHistoryNest2[0]						:= stCycleDataNest2;
	
END_IF
END_ACTION

ACTION d_ACT_IO:
//INPUTS

bPartPresentNest1					:= dw_T08_EL1809.iPartPresentNest1;
bPartPresentNest2					:= dw_T08_EL1809.iPartPresentNest2;

rRejectSensor( CLK := dw_T08_EL1809.iRejectSensor);

bDoorClosingFlag					:= (eCycleState = E_General_ProcessCycle.CLOSE_PROCESS_DOOR) OR (eCycleState = E_General_ProcessCycle.WAIT_CLOSE_PROCESS_DOOR) OR
										bDoorClosingInitFlag;
bDoorOpeningFlag					:= eCycleState = E_General_ProcessCycle.OPEN_PROCESS_DOOR;

bProcessDoorClosedConditionFlag		:= eCycleState = E_General_ProcessCycle.PROCESS_FLAGS_DEFINITIONS OR
										eCycleState = E_General_ProcessCycle.EXTEND_PROCESS_CYLINDER OR
										eCycleState = E_General_ProcessCycle.LEAK_TESTS_HEIGHT_TEST OR
										eCycleState = E_General_ProcessCycle.WAIT_LEAK_TEST_HEIGHT_TEST OR
										eCycleState = E_General_ProcessCycle.HEIGHT_TEST OR
										eCycleState = E_General_ProcessCycle.WAIT_HEIGHT_TEST OR
										eCycleState = E_General_ProcessCycle.LEAK_TESTS OR
										eCycleState = E_General_ProcessCycle.WAIT_LEAK_TEST OR
										eCycleState = E_General_ProcessCycle.CAMERA_INSPECTION OR
										eCycleState = E_General_ProcessCycle.WAIT_CAMERA OR
										eCycleState = E_General_ProcessCycle.RESULTS OR
										eCycleState = E_General_ProcessCycle.WAIT_TO_SAVE_DATA OR
										eCycleState = E_General_ProcessCycle.SAVE_DATA OR
										eCycleState = E_General_ProcessCycle.SAVE_DATA2 OR
										eCycleState = E_General_ProcessCycle.CSV_NEST1 OR
										eCycleState = E_General_ProcessCycle.CSV_NEST2 OR
										eCycleState = E_General_ProcessCycle.RETRACT_PROCESS_CYLINDER OR
										eCycleState = E_General_ProcessCycle.WAIT_RETRACT_PROCESS_CYLINDER;
					

										

										
tonTwoHandsSignal( IN := stTwinSAFE.qTwoHandsSafe , PT := stTimers.tTwoHandsSignal);						
				
bTwoHandsSignal						:= tonTwoHandsSignal.Q;

		
dw_T09_EL2809.qIndicatorLED1_Red	:= stCycleDataNest1.bFail;		
dw_T09_EL2809.qIndicatorLED1_Green	:= stCycleDataNest1.bPass;	
dw_T09_EL2809.qIndicatorLED2_Red	:= stCycleDataNest2.bFail;		
dw_T09_EL2809.qIndicatorLED2_Green	:= stCycleDataNest2.bPass;	

IF 	(stMachineStatus.eMachineState = E_MachineState.SYSTEM_AUTO_CYCLE) AND NOT ((eCycleState	= E_General_ProcessCycle.IDLE) OR (eCycleState	= E_General_ProcessCycle.WAIT_REJECT_PART) 
	OR (eCycleState	= E_General_ProcessCycle.NEST_CLEARING) OR (eCycleState	= E_General_ProcessCycle.REJECT_CHUTE_FULL) OR (eCycleState	= E_General_ProcessCycle.PUCK_DEFINITION)) THEN
	

	bPartPresent[0]					:= 	bProcessedPart[0];
	bPartPresent[1]					:= 	bProcessedPart[1];
	
ELSE	
		bPartPresent[0]				:= dw_T08_EL1809.iPartPresentNest1;
		bPartPresent[1]				:= dw_T08_EL1809.iPartPresentNest2;

END_IF

stTwinSAFE.iMachineHoming_Manual	:= 	stMachineStatus.eMachineState = E_MachineState.SAFETY OR
										stMachineStatus.eMachineState = E_MachineState.SYSTEM_INITIALISING OR
										stMachineStatus.eMachineState = E_MachineState.MANUAL_MODE;
END_ACTION

ACTION e_ACT_SafetyProcess:

END_ACTION

END_PROGRAM

// ---- POUs/B_STATIONS/B_5_PUCK_LOCKER/B_5_1_PRG_PuckLocker.TcPOU
PROGRAM B_5_1_PRG_PuckLocker
VAR
	// ============================================================
    // Local process variables
    // ============================================================
    eMode                       : E_PuckLockerMode;

    bPuckPresentRaw             : BOOL;
    bPuckPresent                : BOOL;

    bPuckSensorsMismatchRaw     : BOOL;
    bPuckSensorsMismatch        : BOOL;

    bEnableEmptyPuckBypass      : BOOL;


    // ============================================================
    // Edge detection
    // ============================================================
    rTrigPuckPresent          : R_TRIG;
    fTrigPuckPresent          : F_TRIG;

    rTrigApplyDisposition     : R_TRIG;
    rTrigEmptyPuckBypass      : R_TRIG;
    rTrigAcknowledgeFault     : R_TRIG;


    // ============================================================
    // Timers
    // ============================================================
    tonPuckPresentOnDelay        : TON;
    tonPuckPresentOffDelay       : TON;

    tonPuckMismatchDelay         : TON;
	tonPuckPresentDebounce		 : TON;
	
    tonPinLockDelay              : TON;
	
END_VAR

// =================================================================
// 1. Engineering / HMI configuration
// =================================================================
// eMode should be persistent through your existing GVL_HMI Persistent
// implementation, or copied there from the Engineering page.
// =================================================================
// Puck locker HMI mode selection
// =================================================================


(* Renan Added 10Jul26 - Puck Locker common code *)
IF NOT stMACHINE.bPuckLocker THEN

    eMode := E_PuckLockerMode.Disabled;
    GVL_HMI.stPuckLocker.eMode := eMode;
    GVL_HMI.ePuckLockerMode := eMode;

ELSE

    IF NOT GVL_HMI.bPuckLockerGateEnable THEN
        GVL_HMI.bPuckLockerSkipEnable := FALSE;
    END_IF;

    IF NOT GVL_HMI.bPuckLockerGateEnable THEN

        eMode := E_PuckLockerMode.Disabled;

    ELSIF GVL_HMI.bPuckLockerSkipEnable THEN

        eMode := E_PuckLockerMode.EnabledWithEmptyPuckBypass;

    ELSE

        eMode := E_PuckLockerMode.Enabled;

    END_IF;

    GVL_HMI.ePuckLockerMode := eMode;
    GVL_HMI.stPuckLocker.eMode := eMode;

END_IF;
(*\Renan Added 10Jul26 - Puck Locker common code *)

// Skip option is never allowed while gate is disabled.
IF NOT GVL_HMI.bPuckLockerGateEnable THEN
    GVL_HMI.bPuckLockerSkipEnable := FALSE;
END_IF;

// Convert HMI toggles into the internal locker mode.
IF NOT GVL_HMI.bPuckLockerGateEnable THEN

    eMode := E_PuckLockerMode.Disabled;

ELSIF GVL_HMI.bPuckLockerSkipEnable THEN

    eMode := E_PuckLockerMode.EnabledWithEmptyPuckBypass;

ELSE

    eMode := E_PuckLockerMode.Enabled;

END_IF;

// Keep existing status/interface compatible.
GVL_HMI.ePuckLockerMode := eMode;
GVL_HMI.stPuckLocker.eMode := eMode;


// =================================================================
// 2. Read physical inputs
// =================================================================
GVL_Stations.stPuckLocker.bPuckSensorUp 	:= GVL_IO.dw_T08_EL1809.iPuckSensorUp;
GVL_Stations.stPuckLocker.bPuckSensorDown 	:= GVL_IO.dw_T08_EL1809.iPuckSensorDown;

// =================================================================
// 3. Validate puck presence
// =================================================================
// The puck is considered correctly positioned only when both sensors
// are active simultaneously.
bPuckPresentRaw := GVL_Stations.stPuckLocker.bPuckSensorUp AND GVL_Stations.stPuckLocker.bPuckSensorDown;

GVL_IO.stTwinSAFE.iPuckError := GVL_Stations.stPuckLocker.bUnexpectedRemovalFault;

// One sensor ON and the other OFF may be caused by:
// - puck moving through the sensing area;
// - puck not aligned;
// - puck partially lifted;
// - sensor issue.
bPuckSensorsMismatchRaw :=GVL_Stations.stPuckLocker.bPuckSensorUp XOR GVL_Stations.stPuckLocker.bPuckSensorDown;

// Require both sensors active for 100 ms before confirming puck.
tonPuckPresentOnDelay(IN := bPuckPresentRaw,PT := T#100MS);

// Require both sensors inactive for 100 ms before confirming absence.
tonPuckPresentOffDelay(IN := NOT bPuckPresentRaw,PT := T#100MS);


IF tonPuckPresentOnDelay.Q THEN

    bPuckPresent := TRUE;

ELSIF tonPuckPresentOffDelay.Q THEN

    bPuckPresent := FALSE;

END_IF

// Debounce puck present
tonPuckPresentDebounce(IN := bPuckPresentRaw, PT := T#100MS);

// Debounced puck detection
GVL_Stations.stPuckLocker.bPuckDetected := tonPuckPresentDebounce.Q;

// Keep mismatch indication only after a short delay, so normal puck
// movement does not generate false warnings.
tonPuckMismatchDelay(IN := bPuckSensorsMismatchRaw,PT := T#500MS);

bPuckSensorsMismatch := tonPuckMismatchDelay.Q;

// =================================================================
// 4. Edge detection
// =================================================================
rTrigPuckPresent(CLK := bPuckPresent);

fTrigPuckPresent(CLK := bPuckPresent);

rTrigApplyDisposition(CLK := GVL_Stations.stPuckLocker.bApplyDisposition);

rTrigEmptyPuckBypass(CLK := GVL_HMI.stPuckLocker.bCmdEmptyPuckBypass);

rTrigAcknowledgeFault(CLK := GVL_HMI.stPuckLocker.bCmdAcknowledgeRemovalFault AND bPuckPresent);//Puck present added 

IF NOT bPuckPresent THEN
	
	GVL_HMI.stPuckLocker.bCmdAcknowledgeRemovalFault := FALSE;

END_IF


// =================================================================
// 5. Latch disposition request from MachineCtrl
// =================================================================
// MachineCtrl should write these values once, after both final nest
// results are known:
//
// PASS / PASS:
// nRequestedRelease := 2;
// nRequestedRemoval := 0;
//
// PASS / FAIL or FAIL / PASS:
// nRequestedRelease := 1;
// nRequestedRemoval := 0;
//
// FAIL / FAIL:
// nRequestedRelease := 0;
// nRequestedRemoval := 1;
//
// bApplyDisposition := TRUE;
IF rTrigApplyDisposition.Q THEN

    IF GVL_Stations.stPuckLocker.nRequestedRelease > USINT#2 THEN
        GVL_Stations.stPuckLocker.nPucksAllowedToPass := USINT#2;
    ELSE
        GVL_Stations.stPuckLocker.nPucksAllowedToPass :=
            GVL_Stations.stPuckLocker.nRequestedRelease;
    END_IF

    GVL_Stations.stPuckLocker.bDispositionPending := TRUE;
    GVL_Stations.stPuckLocker.bApplyDisposition := FALSE;

END_IF


// =================================================================
// 6. Default values
// =================================================================
GVL_Stations.stPuckLocker.bRemovalAllowed := FALSE;
bEnableEmptyPuckBypass := FALSE;

tonPinLockDelay(IN := GVL_Stations.stPuckLocker.eState = E_PuckLockerState.LockingPuck AND bPuckPresent, PT := T#300MS);

IF stMachineStatus.bInitialising OR stMachineStatus.eMachineState = E_MachineState.SYSTEM_INITIALISING THEN

    f_ACT_ResetPuckLocker();
    RETURN;

END_IF

// =================================================================
// 8. Main Puck Locker State Machine
// =================================================================
CASE GVL_Stations.stPuckLocker.eState OF


    // ------------------------------------------------------------
    // Locker disabled.
    // Pin remains down and does not interfere with puck movement.
    // ------------------------------------------------------------
    E_PuckLockerState.Disabled:

        GVL_Stations.stPuckLocker.bPinCommandUp := FALSE;

        GVL_Stations.stPuckLocker.bPuckLocked := FALSE;
        GVL_Stations.stPuckLocker.bUnexpectedRemovalFault := FALSE;

        GVL_Stations.stPuckLocker.nPucksAllowedToPass := 0;
        GVL_Stations.stPuckLocker.nPucksToRemove := 0;

        GVL_Stations.stPuckLocker.bDispositionPending := FALSE;
        GVL_Stations.stPuckLocker.bDispositionHandled := FALSE;

        IF eMode <> E_PuckLockerMode.Disabled THEN

            GVL_Stations.stPuckLocker.eState := E_PuckLockerState.WaitingForPuck;

        END_IF


    // ------------------------------------------------------------
    // Pin remains down. Wait for a properly centred puck.
    // ------------------------------------------------------------
    E_PuckLockerState.WaitingForPuck:

        GVL_Stations.stPuckLocker.bPinCommandUp := FALSE;
        GVL_Stations.stPuckLocker.bPuckLocked := FALSE;

        IF eMode = E_PuckLockerMode.Disabled THEN

            GVL_Stations.stPuckLocker.eState := E_PuckLockerState.Disabled;

        ELSIF bPuckPresent
              AND GVL_Stations.stPuckLocker.nPucksAllowedToPass = 0
              AND GVL_Stations.stPuckLocker.nPucksToRemove = 0 THEN

            GVL_Stations.stPuckLocker.eState := E_PuckLockerState.LockingPuck;

        END_IF


    // ------------------------------------------------------------
    // Pin command is up.
    // No physical feedback exists, so locking is accepted after
    // 300 ms while the puck stays detected.
    // ------------------------------------------------------------
    E_PuckLockerState.LockingPuck:

        GVL_Stations.stPuckLocker.bPinCommandUp := TRUE;
		GVL_Stations.stPuckLocker.bPuckLocked := FALSE;
	
		IF eMode = E_PuckLockerMode.Disabled THEN
	
			GVL_Stations.stPuckLocker.eState := E_PuckLockerState.Disabled;
	
		ELSIF NOT bPuckPresent THEN
	
			// Puck was not fully captured yet.
			// Return to waiting state without fault.
			GVL_Stations.stPuckLocker.eState := E_PuckLockerState.WaitingForPuck;
	
		ELSIF tonPinLockDelay.Q THEN
	
			GVL_Stations.stPuckLocker.bPuckLocked := TRUE;
			GVL_Stations.stPuckLocker.eState := E_PuckLockerState.Locked;
	
		END_IF


    // ------------------------------------------------------------
    // Puck captured by locker pin.
    // Wait for process disposition, bypass request or fault.
    // ------------------------------------------------------------
    E_PuckLockerState.Locked:

        GVL_Stations.stPuckLocker.bPinCommandUp := TRUE;
        GVL_Stations.stPuckLocker.bPuckLocked := TRUE;


        // Bypass is only allowed in the configured bypass mode.
        // It is disabled once a process disposition is pending.
        bEnableEmptyPuckBypass := (eMode = E_PuckLockerMode.EnabledWithEmptyPuckBypass) AND NOT GVL_Stations.stPuckLocker.bDispositionPending AND NOT GVL_Stations.stPuckLocker.bUnexpectedRemovalFault;


        // Puck disappeared while pin should have been holding it.
        IF NOT bPuckPresent THEN

            GVL_Stations.stPuckLocker.bUnexpectedRemovalFault := TRUE;
            GVL_Stations.stPuckLocker.eState := E_PuckLockerState.UnexpectedPuckRemovalFault;


        // Empty puck bypass confirmed through HMI.
        ELSIF rTrigEmptyPuckBypass.Q
              AND bEnableEmptyPuckBypass THEN

            GVL_Stations.stPuckLocker.nPucksAllowedToPass := 1;
            GVL_Stations.stPuckLocker.nPucksToRemove := 0;

            GVL_HMI.stPuckLocker.bCmdEmptyPuckBypass := FALSE;

            GVL_Stations.stPuckLocker.eState := E_PuckLockerState.ReleasingPucks;


        // Final disposition received from MachineCtrl.
		ELSIF GVL_Stations.stPuckLocker.bDispositionPending THEN

			GVL_Stations.stPuckLocker.bDispositionPending := FALSE;
		
			// Release is authorised, but the pin must remain up until
			// both nests are empty. This ensures the PASS part was placed
			// back onto the locked puck before it can be released.
			IF GVL_Stations.stPuckLocker.nPucksAllowedToPass > 0 THEN
		
				GVL_Stations.stPuckLocker.eState := E_PuckLockerState.WaitingForNestsEmpty;
		
			END_IF
		END_IF


    E_PuckLockerState.WaitingForNestsEmpty:

		// Keep puck physically locked while either nest still contains
		// a product.
		GVL_Stations.stPuckLocker.bPinCommandUp := TRUE;
		GVL_Stations.stPuckLocker.bPuckLocked := TRUE;
	
		IF NOT bPuckPresent THEN
	
			GVL_Stations.stPuckLocker.bUnexpectedRemovalFault := TRUE;
	
			GVL_Stations.stPuckLocker.eState := E_PuckLockerState.UnexpectedPuckRemovalFault;
	
		ELSIF GVL_Stations.stPuckLocker.bNestsEmpty AND GVL_Stations.stPuckLocker.nPucksAllowedToPass > 0 THEN
	
			GVL_Stations.stPuckLocker.eState := E_PuckLockerState.ReleasingPucks;
	
		END_IF
		
    // ------------------------------------------------------------
    // Pin is down. One or two authorised pucks may pass.
    // A puck is counted when it clears both sensors.
    // ------------------------------------------------------------
    E_PuckLockerState.ReleasingPucks:

        GVL_Stations.stPuckLocker.bPinCommandUp := FALSE;
        GVL_Stations.stPuckLocker.bPuckLocked := FALSE;

        IF fTrigPuckPresent.Q
           AND GVL_Stations.stPuckLocker.nPucksAllowedToPass > 0 THEN

            GVL_Stations.stPuckLocker.nPucksAllowedToPass := GVL_Stations.stPuckLocker.nPucksAllowedToPass - 1;

        END_IF

        // All authorised pucks passed through the locker.
		// Return to rest/waiting state. No timeout is required here.
		IF GVL_Stations.stPuckLocker.nPucksAllowedToPass = 0
		AND NOT bPuckPresent THEN
		
			GVL_Stations.stPuckLocker.eState := E_PuckLockerState.WaitingForPuck;
		
		END_IF


    // ------------------------------------------------------------
    // Puck was removed unexpectedly while locked.
    // Pin stays down for safe recovery.
    //
    // Operator must return the puck to the sensor area and an
    // authorised user must acknowledge the event.
    // ------------------------------------------------------------
    E_PuckLockerState.UnexpectedPuckRemovalFault:

		GVL_Stations.stPuckLocker.bPinCommandUp := FALSE;
		GVL_Stations.stPuckLocker.bPuckLocked := FALSE;
	
		GVL_Stations.stPuckLocker.bUnexpectedRemovalFault := TRUE;
	
		IF eMode = E_PuckLockerMode.Disabled THEN
	
			GVL_Stations.stPuckLocker.eState := E_PuckLockerState.Disabled;
	
		ELSIF bPuckPresent AND rTrigAcknowledgeFault.Q THEN
		
			GVL_HMI.stPuckLocker.bCmdAcknowledgeRemovalFault := FALSE;
			GVL_Stations.stPuckLocker.bUnexpectedRemovalFault := FALSE;
			GVL_Stations.stPuckLocker.eState := E_PuckLockerState.LockingPuck;

		END_IF

END_CASE


// =================================================================
// 8. Write HMI interface
// =================================================================
GVL_HMI.stPuckLocker.bEnableEmptyPuckBypass := bEnableEmptyPuckBypass;

GVL_HMI.stPuckLocker.bPuckDetected := bPuckPresent;

GVL_HMI.stPuckLocker.bPuckLocked := GVL_Stations.stPuckLocker.bPuckLocked;

GVL_HMI.stPuckLocker.bPuckSensorMismatch := bPuckSensorsMismatch;

GVL_HMI.stPuckLocker.bUnexpectedRemovalFault := GVL_Stations.stPuckLocker.bUnexpectedRemovalFault;

GVL_HMI.stPuckLocker.bShowUnexpectedRemovalPopup := GVL_Stations.stPuckLocker.bUnexpectedRemovalFault;

GVL_HMI.stPuckLocker.nPucksAllowedToPass := GVL_Stations.stPuckLocker.nPucksAllowedToPass;


// This can remain FALSE if the HMI itself opens the confirmation
// popup after the operator presses the bypass button.
GVL_HMI.stPuckLocker.bShowEmptyPuckPopup := FALSE;


// =================================================================
// 9. Message generation
// =================================================================
CASE GVL_Stations.stPuckLocker.eState OF

    E_PuckLockerState.Disabled:
        GVL_Stations.stPuckLocker.sMessage := 'PUCK LOCKER DISABLED';

    E_PuckLockerState.WaitingForPuck:
        GVL_Stations.stPuckLocker.sMessage := 'WAITING FOR PUCK';

    E_PuckLockerState.LockingPuck:
        GVL_Stations.stPuckLocker.sMessage := 'LOCKING PUCK';

    E_PuckLockerState.Locked:
        GVL_Stations.stPuckLocker.sMessage := 'PUCK LOCKED';
		
	E_PuckLockerState.WaitingForNestsEmpty:
    	GVL_Stations.stPuckLocker.sMessage := 'UNLOAD BOTH NESTS BEFORE PUCK RELEASE';

    E_PuckLockerState.ReleasingPucks:
        GVL_Stations.stPuckLocker.sMessage := 'PUCK RELEASE IN PROGRESS';

    E_PuckLockerState.UnexpectedPuckRemovalFault:
        GVL_Stations.stPuckLocker.sMessage := 'PUCK REMOVED WHILE LOCKED. RETURN PUCK AND ACKNOWLEDGE.';

END_CASE

GVL_HMI.stPuckLocker.sMessage := GVL_Stations.stPuckLocker.sMessage;

// =================================================================
// 10. Physical output
// =================================================================
// This PRG must remain the only writer of the locker output.
GVL_IO.dw_T09_EL2809.qPuckLockerPinCommand := NOT GVL_Stations.stPuckLocker.bPinCommandUp;

ACTION f_ACT_ResetPuckLocker:
// ================================================================
// f_ACT_ResetPuckLocker
//
// Safe reset of puck locker internal state.
// Pin is commanded to release position.
// ================================================================

GVL_Stations.stPuckLocker.eState := E_PuckLockerState.WaitingForPuck;

GVL_Stations.stPuckLocker.bPinCommandUp := FALSE;
GVL_Stations.stPuckLocker.bPuckLocked := FALSE;
GVL_Stations.stPuckLocker.bRemovalAllowed := FALSE;

GVL_Stations.stPuckLocker.bUnexpectedRemovalFault := FALSE;

GVL_Stations.stPuckLocker.nPucksAllowedToPass := 0;
GVL_Stations.stPuckLocker.nPucksToRemove := 0;

GVL_Stations.stPuckLocker.nRequestedRelease := 0;
GVL_Stations.stPuckLocker.nRequestedRemoval := 0;

GVL_Stations.stPuckLocker.bApplyDisposition := FALSE;
GVL_Stations.stPuckLocker.bDispositionPending := FALSE;
GVL_Stations.stPuckLocker.bDispositionHandled := FALSE;

GVL_HMI.stPuckLocker.bCmdEmptyPuckBypass := FALSE;
GVL_HMI.stPuckLocker.bCmdAcknowledgeRemovalFault := FALSE;

GVL_HMI.stPuckLocker.bEnableEmptyPuckBypass := FALSE;
GVL_HMI.stPuckLocker.bShowUnexpectedRemovalPopup := FALSE;
GVL_HMI.stPuckLocker.bShowEmptyPuckPopup := FALSE;

GVL_HMI.stPuckLocker.bUnexpectedRemovalFault := FALSE;
GVL_HMI.stPuckLocker.nPucksAllowedToPass := 0;
GVL_HMI.stPuckLocker.sMessage := '';
END_ACTION

END_PROGRAM

// ---- POUs/D_CSV/D_1_PRG_CycleDataCSV.TcPOU
PROGRAM D_1_PRG_CycleDataCSV
VAR_INPUT
	
	stCycleDataNest1		: ST_CycleData;
	stCycleDataNest2		: ST_CycleData;
	bWriteNest1				: BOOL;
	bWriteNest2				: BOOL;
	
	
END_VAR
VAR_OUTPUT
	
	bCSVDone				: BOOL;
	bReady					: BOOL;
	
END_VAR
VAR
	sFileName		: T_MaxString := 'C:\Temp\USW_STN13_#date#.csv';(* CSV destination file path and name *)
	sCSVLine		: T_MaxString := '#1#;#2#;#3#;#4#;#5#;#6#;#7#;#8#;#9#,#10#,#11#,#12#,#13#$L';(*1-Nest; 2-General result; 3-Height check; 4-Camera result; 5-Leak tester result; 6-Distance1; 7-Distance2; 8-Distance3; 9-Setpoint 1 10-Setpoint 2 12-Setpoint 3 11-date 3 13-time 3*)
	bBusy			: BOOL;
	bError			: BOOL;
	nErrId			: UDINT;
	hFile			: UINT		:= 0;
	step			: DWORD 	:= 0;
	fbFileOpen		: FB_FileOpen;(* Opens file *)
	fbFileClose		: FB_FileClose;(* Closes file *)
	fbFilePuts		: FB_FilePuts;(* Writes one record (line) *)
	
	done: BOOL;
	
	f1_Nest			: STRING;
	f2_GeneralResult: STRING;
	f3_HeightResult	: STRING;
	f4_CameraResult	: STRING;
	f5_LeakTesterResult	: STRING;
	f6_Distance1	: STRING;
	f7_Distance2	: STRING;
	f8_Distance3	: STRING;
	f9_Setpoint1	: STRING;
	f10_Setpoint2	: STRING;
	f11_Setpoint3	: STRING;
	f12_RawValue1	: STRING;
	f13_RawValue2	: STRING;
	f14_RawValue3	: STRING;
	f15_RawValue4	: STRING;
	f16_Date		: STRING;
	f17_Time		: STRING;
	
	bWritingFirstRow : BOOL;
	bWrite			: BOOL;
	rWriteNest1		: R_TRIG;
	rWriteNest2		: R_TRIG;
	
	rError			: R_TRIG;
	
END_VAR



IF 	step = 0 THEN
	
		bReady		:= TRUE;

ELSE 	bReady		:= FALSE;
END_IF

CASE step OF
	0:	(* Wait for rising edge at bWrite variable *)
		bCSVDone	:= FALSE;
		IF bWrite	 THEN
			
			bWrite	:= FALSE;
			bBusy 	:= TRUE;
			bError	:= FALSE;
			nErrId	:= 0;
			hFile	:= 0;
			step 	:= 1;
			
		END_IF
		
	1:	(* Open source file *)
		fbFileOpen(  bExecute := FALSE  );
		fbFileOpen( sNetId := NetAmsIdLocal, 
					sPathName := sFileName, 
					nMode := FOPEN_MODEAPPEND OR FOPEN_MODETEXT,
					ePath := PATH_GENERIC, 
					bExecute := TRUE );
		step := 2;
	
	2:(* Wait until open not busy *)
		fbFileOpen( bExecute := FALSE, bError => bError, nErrID => nErrID, hFile => hFile );
		IF NOT fbFileOpen.bBusy THEN
			IF NOT fbFileOpen.bError THEN
				step := 3;
			ELSE(* Error: file not found? *)
				step := 100;
			END_IF
		END_IF

	3:(* Convert one PLC record to CSV format *)
		
		FindAndReplace(pSrcString:= ADR(sCSVLine), pDeleteString:= ADR('#1#'), pInsertString:= ADR(f1_Nest), pDstString:= ADR(sCSVLine), nDstSize:= SIZEOF(sCSVLine));
		FindAndReplace(pSrcString:= ADR(sCSVLine), pDeleteString:= ADR('#2#'), pInsertString:= ADR(f2_GeneralResult), pDstString:= ADR(sCSVLine), nDstSize:= SIZEOF(sCSVLine));
		FindAndReplace(pSrcString:= ADR(sCSVLine), pDeleteString:= ADR('#3#'), pInsertString:= ADR(f3_HeightResult), pDstString:= ADR(sCSVLine), nDstSize:= SIZEOF(sCSVLine));
		FindAndReplace(pSrcString:= ADR(sCSVLine), pDeleteString:= ADR('#4#'), pInsertString:= ADR(f4_CameraResult), pDstString:= ADR(sCSVLine), nDstSize:= SIZEOF(sCSVLine));
		FindAndReplace(pSrcString:= ADR(sCSVLine), pDeleteString:= ADR('#5#'), pInsertString:= ADR(f5_LeakTesterResult), pDstString:= ADR(sCSVLine), nDstSize:= SIZEOF(sCSVLine));
		FindAndReplace(pSrcString:= ADR(sCSVLine), pDeleteString:= ADR('#6#'), pInsertString:= ADR(f6_Distance1), pDstString:= ADR(sCSVLine), nDstSize:= SIZEOF(sCSVLine));
		FindAndReplace(pSrcString:= ADR(sCSVLine), pDeleteString:= ADR('#7#'), pInsertString:= ADR(f7_Distance2), pDstString:= ADR(sCSVLine), nDstSize:= SIZEOF(sCSVLine));
		FindAndReplace(pSrcString:= ADR(sCSVLine), pDeleteString:= ADR('#8#'), pInsertString:= ADR(f8_Distance3), pDstString:= ADR(sCSVLine), nDstSize:= SIZEOF(sCSVLine));
		FindAndReplace(pSrcString:= ADR(sCSVLine), pDeleteString:= ADR('#9#'), pInsertString:= ADR(f9_Setpoint1), pDstString:= ADR(sCSVLine), nDstSize:= SIZEOF(sCSVLine));
		FindAndReplace(pSrcString:= ADR(sCSVLine), pDeleteString:= ADR('#10#'), pInsertString:= ADR(f10_Setpoint2), pDstString:= ADR(sCSVLine), nDstSize:= SIZEOF(sCSVLine));
		FindAndReplace(pSrcString:= ADR(sCSVLine), pDeleteString:= ADR('#11#'), pInsertString:= ADR(f11_Setpoint3), pDstString:= ADR(sCSVLine), nDstSize:= SIZEOF(sCSVLine));
		FindAndReplace(pSrcString:= ADR(sCSVLine), pDeleteString:= ADR('#12#'), pInsertString:= ADR(f12_RawValue1), pDstString:= ADR(sCSVLine), nDstSize:= SIZEOF(sCSVLine));
		FindAndReplace(pSrcString:= ADR(sCSVLine), pDeleteString:= ADR('#13#'), pInsertString:= ADR(f13_RawValue2), pDstString:= ADR(sCSVLine), nDstSize:= SIZEOF(sCSVLine));
		FindAndReplace(pSrcString:= ADR(sCSVLine), pDeleteString:= ADR('#14#'), pInsertString:= ADR(f14_RawValue3), pDstString:= ADR(sCSVLine), nDstSize:= SIZEOF(sCSVLine));
		FindAndReplace(pSrcString:= ADR(sCSVLine), pDeleteString:= ADR('#15#'), pInsertString:= ADR(f15_RawValue4), pDstString:= ADR(sCSVLine), nDstSize:= SIZEOF(sCSVLine));	
		FindAndReplace(pSrcString:= ADR(sCSVLine), pDeleteString:= ADR('#16#'), pInsertString:= ADR(f16_Date), pDstString:= ADR(sCSVLine), nDstSize:= SIZEOF(sCSVLine));
		FindAndReplace(pSrcString:= ADR(sCSVLine), pDeleteString:= ADR('#17#'), pInsertString:= ADR(f17_Time), pDstString:= ADR(sCSVLine), nDstSize:= SIZEOF(sCSVLine));
		done:=TRUE;
		
		IF done THEN
			step := 4;
			done := FALSE;
		ELSE
			step := 3;
		END_IF
		
		
	4:	(* Write single text line *)
		fbFilePuts( bExecute := FALSE );
		fbFilePuts( sNetId := '', 
					hFile := hFile, 
					sLine := sCSVLine, 
					bExecute := TRUE );
		step := 5;

	5:(* Wait until write not busy *)
		fbFilePuts( bExecute := FALSE, bError => bError, nErrID => nErrID );
		IF NOT fbFilePuts.bBusy THEN
			IF NOT fbFilePuts.bError THEN
				step := 10;
			ELSE(* Error *)
				step := 100;
			END_IF
		END_IF

	10:	(* Close source file *)
		fbFileClose( bExecute := FALSE );
		fbFileClose( sNetId := '', hFile := hFile, bExecute := TRUE );
		sCSVLine:= '#1#;#2#;#3#;#4#;#5#;#6#;#7#;#8#;#9#,#10#,#11#,#12#,#13#,#14#,#15#,#16#,#17#$L';
		step := 11;

	11:(* Wait until close not busy *)
		fbFileClose( bExecute := FALSE, bError => bError, nErrID => nErrID );
		IF ( NOT fbFileClose.bBusy ) THEN
			bWritingFirstRow	:= FALSE;
			
			hFile := 0;
			step := 100;
		END_IF

	100: (* Error or ready step => cleanup *)
		IF ( hFile <> 0 ) THEN
			step := 10; (* Close the source file *)
		ELSE
			bBusy := FALSE;
			step := 0;	(* Ready *)
			bCSVDone	:= TRUE;
		END_IF

END_CASE

IF (lastDateCSV <> sSystemDate) AND NOT dw_T04_EL1918.iResetButton	 THEN
lastDateCSV:= sSystemDate;
sFileName:= 'C:\Users\Administrator\Desktop\csv\CycleData_#date#.csv';
FindAndReplace(pSrcString:= ADR(sFileName), pDeleteString:= ADR('#date#'), pInsertString:= ADR(lastDateCSV), pDstString:= ADR(sFileName), nDstSize:= SIZEOF(sFileName));

f1_Nest			:= 'NEST';
f2_GeneralResult:= 'GENERAL RESULTS';
f3_HeightResult	:= 'HEIGHT CHECK RESULTS';
f4_CameraResult	:= 'CAMERA RESULTS';
f5_LeakTesterResult	:= 'LEAK TESTER RESULTS';
f6_Distance1	:= 'DISTANCE 1';
f7_Distance2	:= 'DISTANCE 2';
f8_Distance3	:= 'DISTANCE 3';
f9_Setpoint1	:= 'SETPOINT 1';
f10_Setpoint2	:= 'SETPOINT 2';
f11_Setpoint3	:= 'SETPOINT 3';
f12_RawValue1	:= 'PROBE POSITION 1';
f13_RawValue2	:= 'PROBE POSITION 2';
f14_RawValue3	:= 'PROBE POSITION 3';
f15_RawValue4	:= 'PROBE POSITION 4';
f16_Date		:= 'DATE';
f17_Time		:= 'TIME';
bWrite			:= TRUE;
bWritingFirstRow	:= TRUE;

END_IF

IF NOT bWritingFirstRow THEN
	ACT_LinkingVariables();
END_IF

rError(CLK := bError);

bCSVError		:= rError.Q;

IF bWritingFirstRow AND dw_T04_EL1918.iResetButton THEN
	
	lastDateCSV			:= '0';
	bCSVError			:= FALSE;			

END_IF

ACTION ACT_LinkingVariables:
rWriteNest1( CLK := bWriteNest1);
rWriteNest2( CLK := bWriteNest2);

IF rWriteNest1.Q THEN
	
	f1_Nest			:= INT_TO_STRING(stCycleDataNest1.nNest);
	f2_GeneralResult:= stCycleDataNest1.sGeneralResult;
	f3_HeightResult	:= stCycleDataNest1.sHeightTestResult;
	f4_CameraResult	:= stCycleDataNest1.sCameraResult;
	f5_LeakTesterResult	:= stCycleDataNest1.sLeakTesterResult;
	f6_Distance1	:= stCycleDataNest1.sDistance1;
	f7_Distance2	:= stCycleDataNest1.sDistance2;
	f8_Distance3	:= stCycleDataNest1.sDistance3;
	f9_Setpoint1	:= stCycleDataNest1.sSetpoint1;
	f10_Setpoint2	:= stCycleDataNest1.sSetpoint2;
	f11_Setpoint3	:= stCycleDataNest1.sSetpoint3;
	f12_RawValue1	:= REAL_TO_STRING(stCycleDataNest1.HeightTest_anRawMeasurement[1]);
	f13_RawValue2	:= REAL_TO_STRING(stCycleDataNest1.HeightTest_anRawMeasurement[2]);
	f14_RawValue3	:= REAL_TO_STRING(stCycleDataNest1.HeightTest_anRawMeasurement[3]);
	f15_RawValue4	:= REAL_TO_STRING(stCycleDataNest1.HeightTest_anRawMeasurement[4]);
	f16_Date		:= stCycleDataNest1.sDate;
	f17_Time		:= stCycleDataNest1.sTime;
	
	bWrite			:= TRUE;

ELSIF rWriteNest2.Q THEN
	
	f1_Nest			:= INT_TO_STRING(stCycleDataNest2.nNest);
	f2_GeneralResult:= stCycleDataNest2.sGeneralResult;
	f3_HeightResult	:= stCycleDataNest2.sHeightTestResult;
	f4_CameraResult	:= stCycleDataNest2.sCameraResult;
	f5_LeakTesterResult	:= stCycleDataNest2.sLeakTesterResult;
	f6_Distance1	:= stCycleDataNest2.sDistance1;
	f7_Distance2	:= stCycleDataNest2.sDistance2;
	f8_Distance3	:= stCycleDataNest2.sDistance3;
	f9_Setpoint1	:= stCycleDataNest2.sSetpoint1;
	f10_Setpoint2	:= stCycleDataNest2.sSetpoint2;
	f11_Setpoint3	:= stCycleDataNest2.sSetpoint3;
	f12_RawValue1	:= REAL_TO_STRING(stCycleDataNest2.HeightTest_anRawMeasurement[1]);
	f13_RawValue2	:= REAL_TO_STRING(stCycleDataNest2.HeightTest_anRawMeasurement[2]);
	f14_RawValue3	:= REAL_TO_STRING(stCycleDataNest2.HeightTest_anRawMeasurement[3]);
	f15_RawValue4	:= REAL_TO_STRING(stCycleDataNest2.HeightTest_anRawMeasurement[4]);
	f16_Date		:= stCycleDataNest2.sDate;
	f17_Time		:= stCycleDataNest2.sTime;
	
	bWrite			:= TRUE;
	
END_IF
END_ACTION

END_PROGRAM
